// TIA Portal V18 export
TYPE "UDT_BoilersSummaryAlarms"
// stored: IsFailsafeCompliant false
   STRUCT
      BlockingAlarm : Array[1..2] of Bool;
   END_STRUCT;
END_TYPE
